FUNCTION F_Settings_Row_Insert : BOOL
VAR_IN_OUT
	aSettings	: ARRAY[*] OF ST_Data_Item; /// settings structure
END_VAR
VAR_INPUT
	nPlace				:INT;
	//stGroup				:ST_Text;
	//stName				:ST_Text;
	//stUnit				:ST_Text;
	//eDataType			:E_DataType;
END_VAR
VAR
	nn	: DINT;
END_VAR

IF (nPlace < LOWER_BOUND(aSettings,1)) OR (nPlace > UPPER_BOUND(aSettings,1)) THEN
	RETURN;
END_IF

//Check Array Size

FOR nn:= (UPPER_BOUND(aSettings,1)-1) TO  MAX(LOWER_BOUND(aSettings,1),nPlace) by -1 DO
	MEMCPY(ADR(aSettings[nn+1]),ADR(aSettings[nn]),SIZEOF(aSettings[nn+1])); (*set  zero*)		
END_FOR
MEMSET(ADR(aSettings[nPlace]),0,SIZEOF(aSettings[nPlace])); (*set  zero*)

END_FUNCTION

(* stored: Version 1.1.0.1, ProductVersion 3.1.4024.11
   POU F_Settings_Row_Insert: Id {c59076d0-6c22-4b45-995a-5a3cc4ca7c93}, SpecialFunc None *)
